(* Schneider Machine Expert - Basic project PartMotor_Felipe_V1_2024_09_26, file version 2.9.0.0 *)
(* CompanyInformations: City=Videira, State=Santa Catarina, Country=Brasil *)
(* ProjectInformations: Name=Projeto_Automacao *)
(* UserInformations: LastName=Biava Favarin, FirstName=Felipe, Email=felipebfavarin@gmail.com, City=Videira, Country=Brasil *)

HARDWARE
  Cpu 0: TM221CE24R
  EthernetConfiguration: NetworkName=M221, IpAllocationMode=FixedAddress, IpAddress=0.0.0.0, SubnetMask=0.0.0.0
  SerialLineConfiguration: Baud=Baud19200, Parity=ParityEven, DataBits=DataBits8, StopBits=StopBits1, PhysicalMedium=PhysicalMediumRs485, TransmissionMode=TransmissionModeModbusRtu, SlaveId=1, Addressing=SlaveAddressing
  MastTask: UsePeriodScanMode=false, PeriodScan=100
  FastTask: Period=255
  CpuBehavior: StartingMode=StartAsPreviousState, AutoSaveRamOnEeprom=true, WatchdogPeriod=250

SYMBOLS  (address, symbol, comment, settings)
  %M0       AUX_PAI_EMERG_ATUA  "auxiliar comando emergencial painel para atuar"
  %M1       AUX_PAI_EMERG_DESA
  %M2       AUX_PAI_LOCA
  %M3       AUX_PAI_REMO
  %M4       AUX_PAI_MOT1_LIGA
  %M5       AUX_PAI_MOT1_DESL
  %M6       AUX_PAI_MOT2_LIGA
  %M7       AUX_PAI_MOT2_DESL
  %M8       MOT1_LIGA_LOCA
  %M9       MOT1_DESL_LOCA
  %M10      MOT2_LIGA_LOCA
  %M11      MOT2_DESL_LOCA
  %M12      INI_REMO
  %M13      FIM_REMO
  %M20      FT_MOT1_LIGA
  %M21      FT_MOT2_LIGA
  %M22      FIM_CIC  "Fim dos Ciclos"
  %M30      MODO_LOCA  "Modo Local"
  %M32      MODO_REMO  "Modo Remoto"
  %M51      HAB_MOT1
  %M52      HAB_MOT2
  %M100     IHM_CMD_INICIO
  %M101     IHM_CMD_FIM
  %MW1      DISP_TEMP1
  %MW3      DISP_TEMP2
  %TM0      TEMP_MOT1  [Preset=10, Base=OneSecond]
  %TM1      TEMP_MOT2  [Preset=15, Base=OneSecond]
  %C0       CON_CIC  [Preset=3]
  %I0.0     CMD_PAI_EMER_ATUA
  %I0.1     CMD_PAI_EMER_DESA
  %I0.2     CMD_PAI_LOCA
  %I0.3     CMD_PAI_REMO
  %I0.4     CMD_PAI_MOT1_LIGA
  %I0.5     CMD_PAI_MOT1_DESL
  %I0.6     CMD_PAI_MOT2_LIGA
  %I0.7     CMD_PAI_MOT2_DESL
  %Q0.1     MOT1
  %Q0.2     MOT2

POU Novo POU
  (* SectionNumber=1 *)

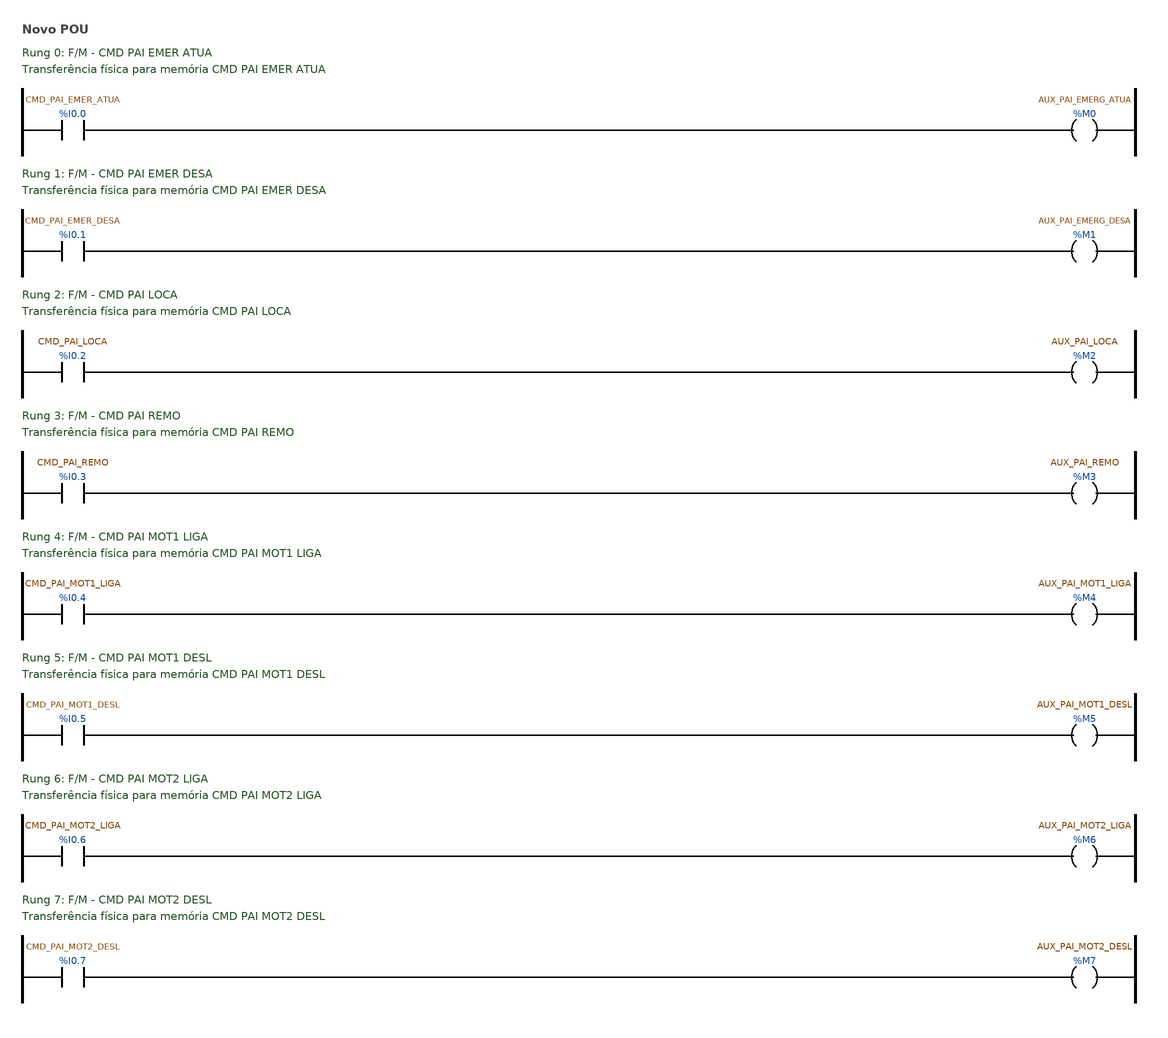

// Rung 0: F/M - CMD PAI EMER ATUA
// Transferência física para memória CMD PAI EMER ATUA
  LD %I0.0                (* CMD_PAI_EMER_ATUA *)
  ST %M0                  (* AUX_PAI_EMERG_ATUA *)
  // as ST:
  //   AUX_PAI_EMERG_ATUA := CMD_PAI_EMER_ATUA;

// Rung 1: F/M - CMD PAI EMER DESA
// Transferência física para memória CMD PAI EMER DESA
  LD %I0.1                (* CMD_PAI_EMER_DESA *)
  ST %M1                  (* AUX_PAI_EMERG_DESA *)
  // as ST:
  //   AUX_PAI_EMERG_DESA := CMD_PAI_EMER_DESA;

// Rung 2: F/M - CMD PAI LOCA
// Transferência física para memória CMD PAI LOCA
  LD %I0.2                (* CMD_PAI_LOCA *)
  ST %M2                  (* AUX_PAI_LOCA *)
  // as ST:
  //   AUX_PAI_LOCA := CMD_PAI_LOCA;

// Rung 3: F/M - CMD PAI REMO
// Transferência física para memória CMD PAI REMO
  LD %I0.3                (* CMD_PAI_REMO *)
  ST %M3                  (* AUX_PAI_REMO *)
  // as ST:
  //   AUX_PAI_REMO := CMD_PAI_REMO;

// Rung 4: F/M - CMD PAI MOT1 LIGA
// Transferência física para memória CMD PAI MOT1 LIGA
  LD %I0.4                (* CMD_PAI_MOT1_LIGA *)
  ST %M4                  (* AUX_PAI_MOT1_LIGA *)
  // as ST:
  //   AUX_PAI_MOT1_LIGA := CMD_PAI_MOT1_LIGA;

// Rung 5: F/M - CMD PAI MOT1 DESL
// Transferência física para memória CMD PAI MOT1 DESL
  LD %I0.5                (* CMD_PAI_MOT1_DESL *)
  ST %M5                  (* AUX_PAI_MOT1_DESL *)
  // as ST:
  //   AUX_PAI_MOT1_DESL := CMD_PAI_MOT1_DESL;

// Rung 6: F/M - CMD PAI MOT2 LIGA
// Transferência física para memória CMD PAI MOT2 LIGA
  LD %I0.6                (* CMD_PAI_MOT2_LIGA *)
  ST %M6                  (* AUX_PAI_MOT2_LIGA *)
  // as ST:
  //   AUX_PAI_MOT2_LIGA := CMD_PAI_MOT2_LIGA;

// Rung 7: F/M - CMD PAI MOT2 DESL
// Transferência física para memória CMD PAI MOT2 DESL
  LD %I0.7                (* CMD_PAI_MOT2_DESL *)
  ST %M7                  (* AUX_PAI_MOT2_DESL *)
  // as ST:
  //   AUX_PAI_MOT2_DESL := CMD_PAI_MOT2_DESL;

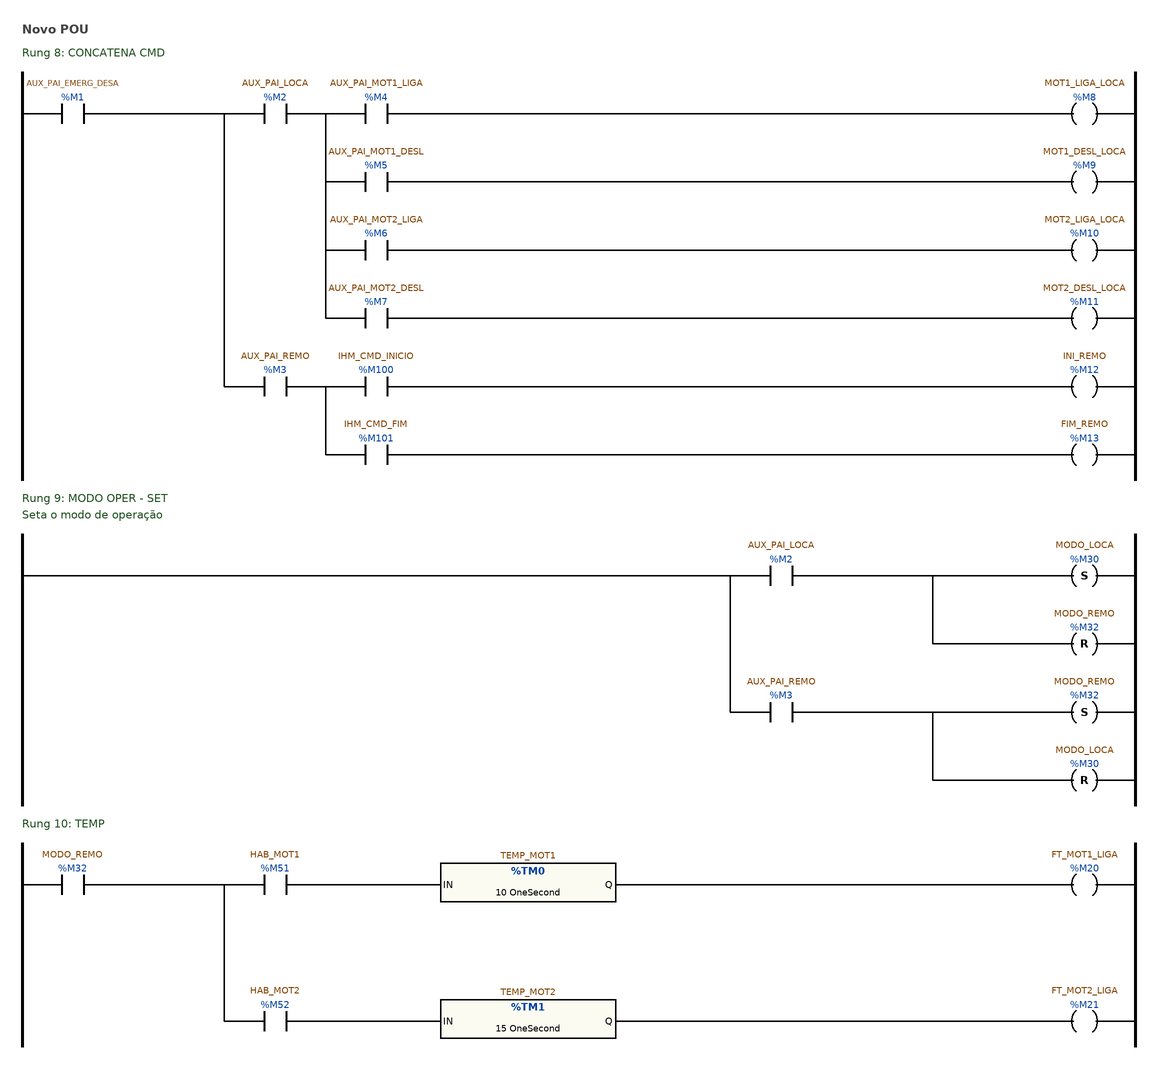

// Rung 8: CONCATENA CMD
  LD %M1                  (* AUX_PAI_EMERG_DESA *)
  MPS
  AND %M2                 (* AUX_PAI_LOCA *)
  MPS
  AND %M4                 (* AUX_PAI_MOT1_LIGA *)
  ST %M8                  (* MOT1_LIGA_LOCA *)
  MRD
  AND %M5                 (* AUX_PAI_MOT1_DESL *)
  ST %M9                  (* MOT1_DESL_LOCA *)
  MRD
  AND %M6                 (* AUX_PAI_MOT2_LIGA *)
  ST %M10                 (* MOT2_LIGA_LOCA *)
  MPP
  AND %M7                 (* AUX_PAI_MOT2_DESL *)
  ST %M11                 (* MOT2_DESL_LOCA *)
  MPP
  AND %M3                 (* AUX_PAI_REMO *)
  MPS
  AND %M100               (* IHM_CMD_INICIO *)
  ST %M12                 (* INI_REMO *)
  MPP
  AND %M101               (* IHM_CMD_FIM *)
  ST %M13                 (* FIM_REMO *)
  // as ST:
  //   MOT1_LIGA_LOCA := AUX_PAI_EMERG_DESA AND AUX_PAI_LOCA AND AUX_PAI_MOT1_LIGA;
  //   MOT1_DESL_LOCA := AUX_PAI_EMERG_DESA AND AUX_PAI_LOCA AND AUX_PAI_MOT1_DESL;
  //   MOT2_LIGA_LOCA := AUX_PAI_EMERG_DESA AND AUX_PAI_LOCA AND AUX_PAI_MOT2_LIGA;
  //   MOT2_DESL_LOCA := AUX_PAI_EMERG_DESA AND AUX_PAI_LOCA AND AUX_PAI_MOT2_DESL;
  //   INI_REMO := AUX_PAI_EMERG_DESA AND AUX_PAI_REMO AND IHM_CMD_INICIO;
  //   FIM_REMO := AUX_PAI_EMERG_DESA AND AUX_PAI_REMO AND IHM_CMD_FIM;

// Rung 9: MODO OPER - SET
// Seta o modo de operação
  LD 1
  MPS
  AND %M2                 (* AUX_PAI_LOCA *)
  S %M30                  (* MODO_LOCA *)
  R %M32                  (* MODO_REMO *)
  MPP
  AND %M3                 (* AUX_PAI_REMO *)
  S %M32                  (* MODO_REMO *)
  R %M30                  (* MODO_LOCA *)
  // as ST:
  //   IF AUX_PAI_LOCA THEN MODO_LOCA := TRUE; END_IF;
  //   IF AUX_PAI_LOCA THEN MODO_REMO := FALSE; END_IF;
  //   IF AUX_PAI_REMO THEN MODO_REMO := TRUE; END_IF;
  //   IF AUX_PAI_REMO THEN MODO_LOCA := FALSE; END_IF;

// Rung 10: TEMP
  LD 1
  MULTIFB
  LD 1
  AND %M32                (* MODO_REMO *)
  ST %MW2009:X0
  BLK %TM0                (* TEMP_MOT1 *)
  LD %MW2009:X0
  AND %M51                (* HAB_MOT1 *)
  IN
  OUT_BLK
  LD Q
  ST %M20                 (* FT_MOT1_LIGA *)
  END_BLK
  BLK %TM1                (* TEMP_MOT2 *)
  LD %MW2009:X0
  AND %M52                (* HAB_MOT2 *)
  IN
  OUT_BLK
  LD Q
  ST %M21                 (* FT_MOT2_LIGA *)
  END_BLK
  MULTIFB
  // as ST:
  //   TEMP_MOT1(IN := MODO_REMO AND HAB_MOT1);
  //   FT_MOT1_LIGA := TEMP_MOT1.Q;
  //   TEMP_MOT2(IN := MODO_REMO AND HAB_MOT2);
  //   FT_MOT2_LIGA := TEMP_MOT2.Q;

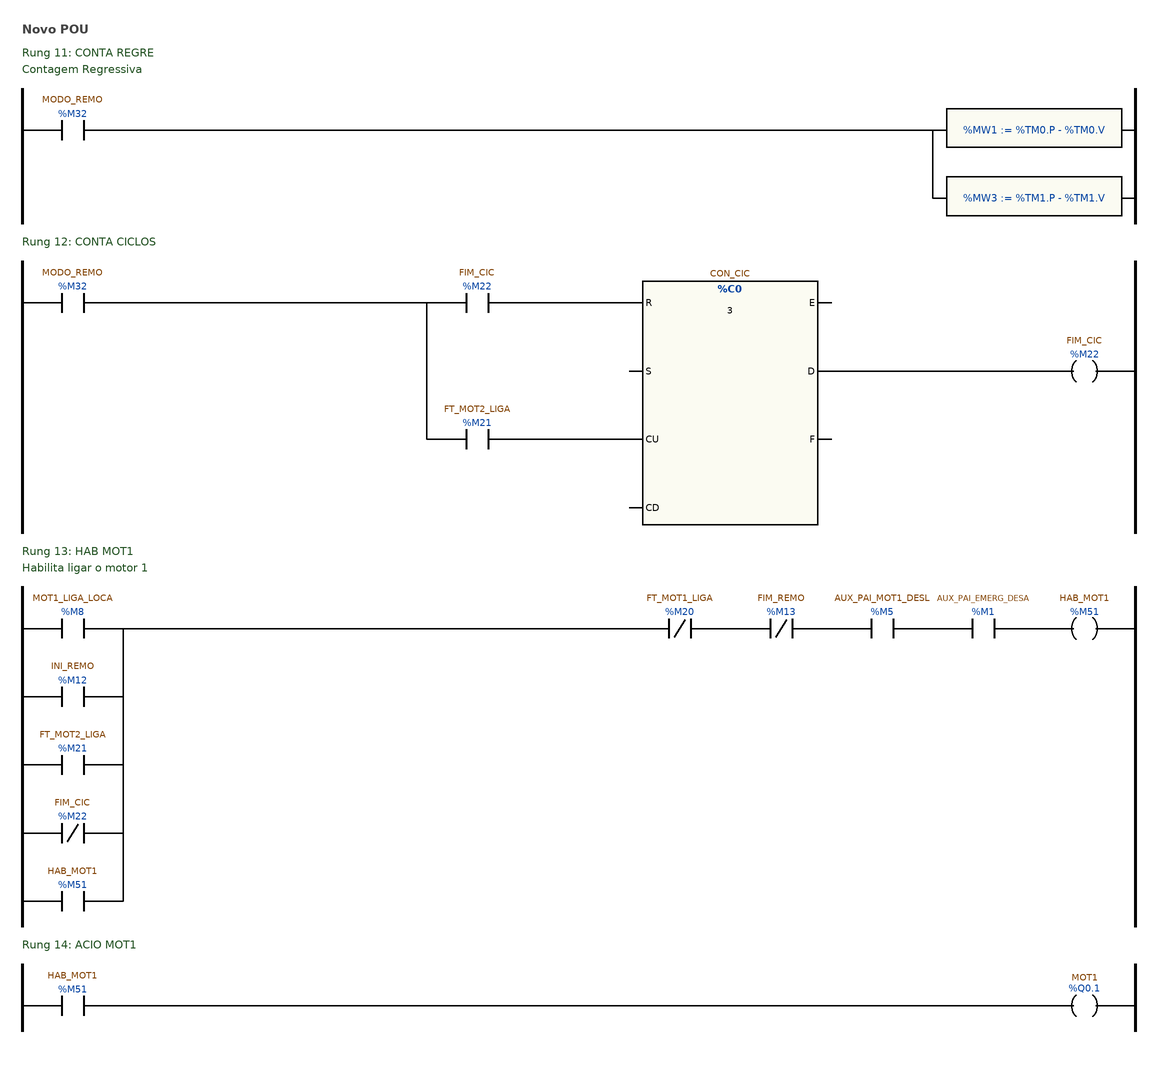

// Rung 11: CONTA REGRE
// Contagem Regressiva
  LD %M32                 (* MODO_REMO *)
  [ %MW1 := %TM0.P - %TM0.V ](* DISP_TEMP1, TEMP_MOT1, TEMP_MOT1 *)
  [ %MW3 := %TM1.P - %TM1.V ](* DISP_TEMP2, TEMP_MOT2, TEMP_MOT2 *)
  // as ST:
  //   IF MODO_REMO THEN DISP_TEMP1 := TEMP_MOT1.P - TEMP_MOT1.V; END_IF;
  //   IF MODO_REMO THEN DISP_TEMP2 := TEMP_MOT2.P - TEMP_MOT2.V; END_IF;

// Rung 12: CONTA CICLOS
  BLK %C0                 (* CON_CIC *)
  LD %M32                 (* MODO_REMO *)
  MPS
  AND %M22                (* FIM_CIC *)
  R
  MPP
  AND %M21                (* FT_MOT2_LIGA *)
  CU
  OUT_BLK
  LD D
  ST %M22                 (* FIM_CIC *)
  END_BLK
  // as ST:
  //   CON_CIC(R := MODO_REMO AND FIM_CIC, CU := MODO_REMO AND FT_MOT2_LIGA);
  //   FIM_CIC := CON_CIC.D;

// Rung 13: HAB MOT1
// Habilita ligar o motor 1
  LD %M8                  (* MOT1_LIGA_LOCA *)
  OR %M12                 (* INI_REMO *)
  OR %M21                 (* FT_MOT2_LIGA *)
  ORN %M22                (* FIM_CIC *)
  OR %M51                 (* HAB_MOT1 *)
  ANDN %M20               (* FT_MOT1_LIGA *)
  ANDN %M13               (* FIM_REMO *)
  AND %M5                 (* AUX_PAI_MOT1_DESL *)
  AND %M1                 (* AUX_PAI_EMERG_DESA *)
  ST %M51                 (* HAB_MOT1 *)
  // as ST:
  //   HAB_MOT1 := (MOT1_LIGA_LOCA OR INI_REMO OR FT_MOT2_LIGA OR NOT FIM_CIC OR HAB_MOT1) AND NOT FT_MOT1_LIGA AND NOT FIM_REMO AND AUX_PAI_MOT1_DESL AND AUX_PAI_EMERG_DESA;

// Rung 14: ACIO MOT1
  LD %M51                 (* HAB_MOT1 *)
  ST %Q0.1                (* MOT1 *)
  // as ST:
  //   MOT1 := HAB_MOT1;

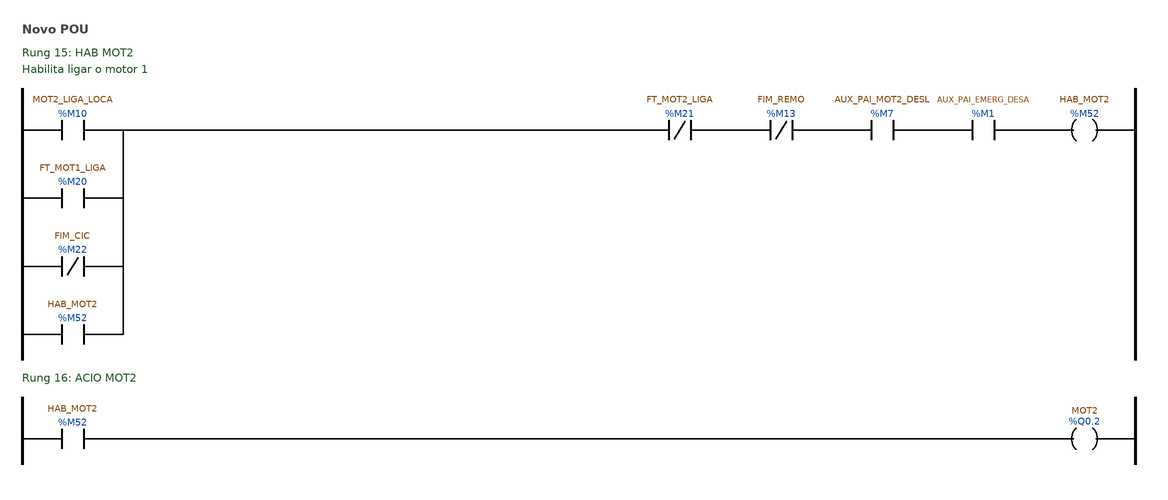

// Rung 15: HAB MOT2
// Habilita ligar o motor 1
  LD %M10                 (* MOT2_LIGA_LOCA *)
  OR %M20                 (* FT_MOT1_LIGA *)
  ORN %M22                (* FIM_CIC *)
  OR %M52                 (* HAB_MOT2 *)
  ANDN %M21               (* FT_MOT2_LIGA *)
  ANDN %M13               (* FIM_REMO *)
  AND %M7                 (* AUX_PAI_MOT2_DESL *)
  AND %M1                 (* AUX_PAI_EMERG_DESA *)
  ST %M52                 (* HAB_MOT2 *)
  // as ST:
  //   HAB_MOT2 := (MOT2_LIGA_LOCA OR FT_MOT1_LIGA OR NOT FIM_CIC OR HAB_MOT2) AND NOT FT_MOT2_LIGA AND NOT FIM_REMO AND AUX_PAI_MOT2_DESL AND AUX_PAI_EMERG_DESA;

// Rung 16: ACIO MOT2
  LD %M52                 (* HAB_MOT2 *)
  ST %Q0.2                (* MOT2 *)
  // as ST:
  //   MOT2 := HAB_MOT2;
